(* IEC 61131-3 sources: Industry-PLC-LLM/data/PLCBEAD_repo/PLCBEAD_PLCEmbed-main/PLC-BEAD/Source/GEB/INT_TO_BCDC, 1 file *)

(* ---- INT_TO_BCDC.ST ---- *)
FUNCTION INT_TO_BCDC:BYTE

	VAR_INPUT
		IN :	INT;
	END_VAR

	INT_TO_BCDC := SHL(INT_TO_BYTE(IN / INT#10),4) OR INT_TO_BYTE(IN MOD INT#10);

END_FUNCTION

PROGRAM program0

	VAR
		IN :	INT;
		OUT : BYTE;
	END_VAR

	OUT := INT_TO_BCDC(IN);

END_PROGRAM
